(* PLC project Unnamed, Unknown Unnamed 1 *)
(* stored: creationDateTime 2025-11-24T11:16:17, modificationDateTime 2025-11-24T18:26:55 *)

PROGRAM Lab2
  VAR
    Potentiometer AT %IW1 : UINT := 0;
    Ljussensor AT %IW2 : UINT;
  END_VAR
  VAR
    S0 : BOOL := False;
    S1 : BOOL := False;
    Light_sample : BOOL := False;
    Poten_sample : BOOL;
    Light_damaged : BOOL := False;
    Poten_damaged : BOOL := False;
    Light_comp : UINT := 32768;
    Damaged : UINT := 0;
    High : UINT := 43690;
    Low : UINT := 21845;
  END_VAR
  VAR
    Relay AT %QX0.0 : BOOL := 0;
  END_VAR
  VAR
    CTU0 : CTU;
    TON0 : TON;
    T50ms : TIME := T#50ms;
    Tick_100ms : BOOL := 0;
    Fifty_ticks : INT := 50;
    TON1 : TON;
    R_TRIG0 : R_TRIG;
    F_TRIG0 : F_TRIG;
  END_VAR
  VAR  (* added by the conversion: wires and edge detectors of the diagram *)
    R_TRIG1 : R_TRIG;
    _GT34_OUT : BOOL;
    _LT35_OUT : BOOL;
    _EQ42_OUT : BOOL;
  END_VAR

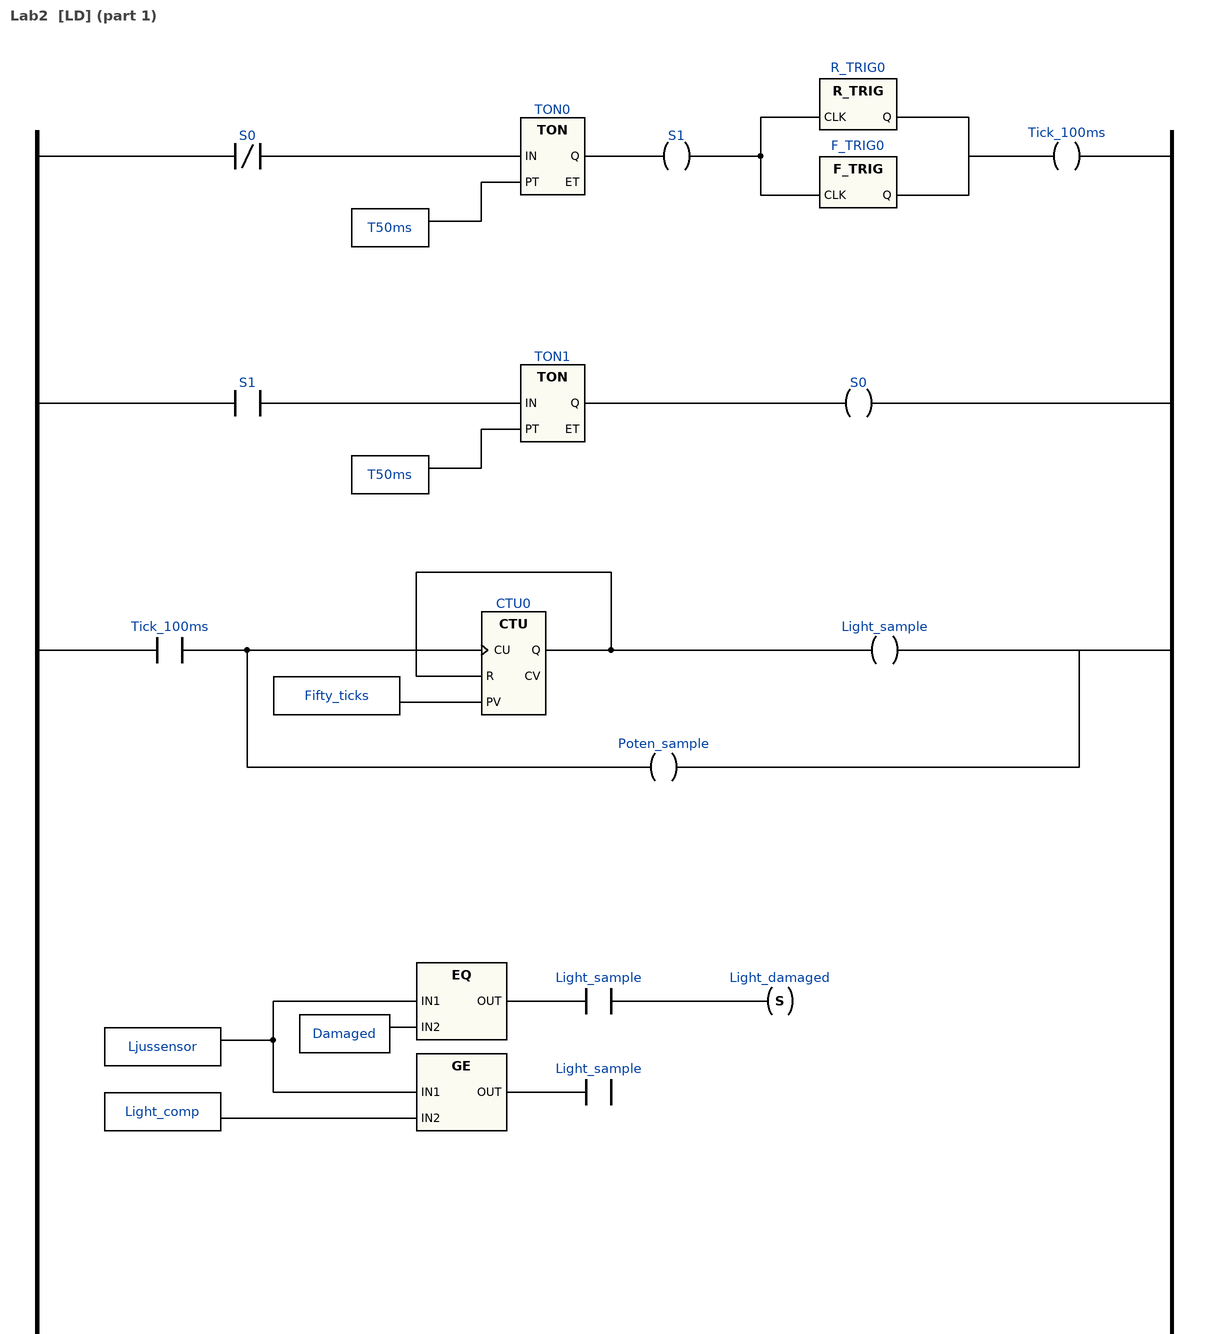
(* LD diagram, written out as Structured Text *)
TON0(IN := NOT S0, PT := T50ms);
R_TRIG0(CLK := TON0.Q);
F_TRIG0(CLK := TON0.Q);
Tick_100ms := R_TRIG0.Q OR F_TRIG0.Q;
R_TRIG1(CLK := Tick_100ms);
CTU0(CU := R_TRIG1.Q, R := CTU0.Q, PV := Fifty_ticks);
Light_sample := CTU0.Q;
TON1(IN := S1, PT := T50ms);
S0 := TON1.Q;
S1 := TON0.Q;
Poten_sample := Tick_100ms;
IF Ljussensor = Damaged AND Light_sample THEN Light_damaged := TRUE; END_IF;
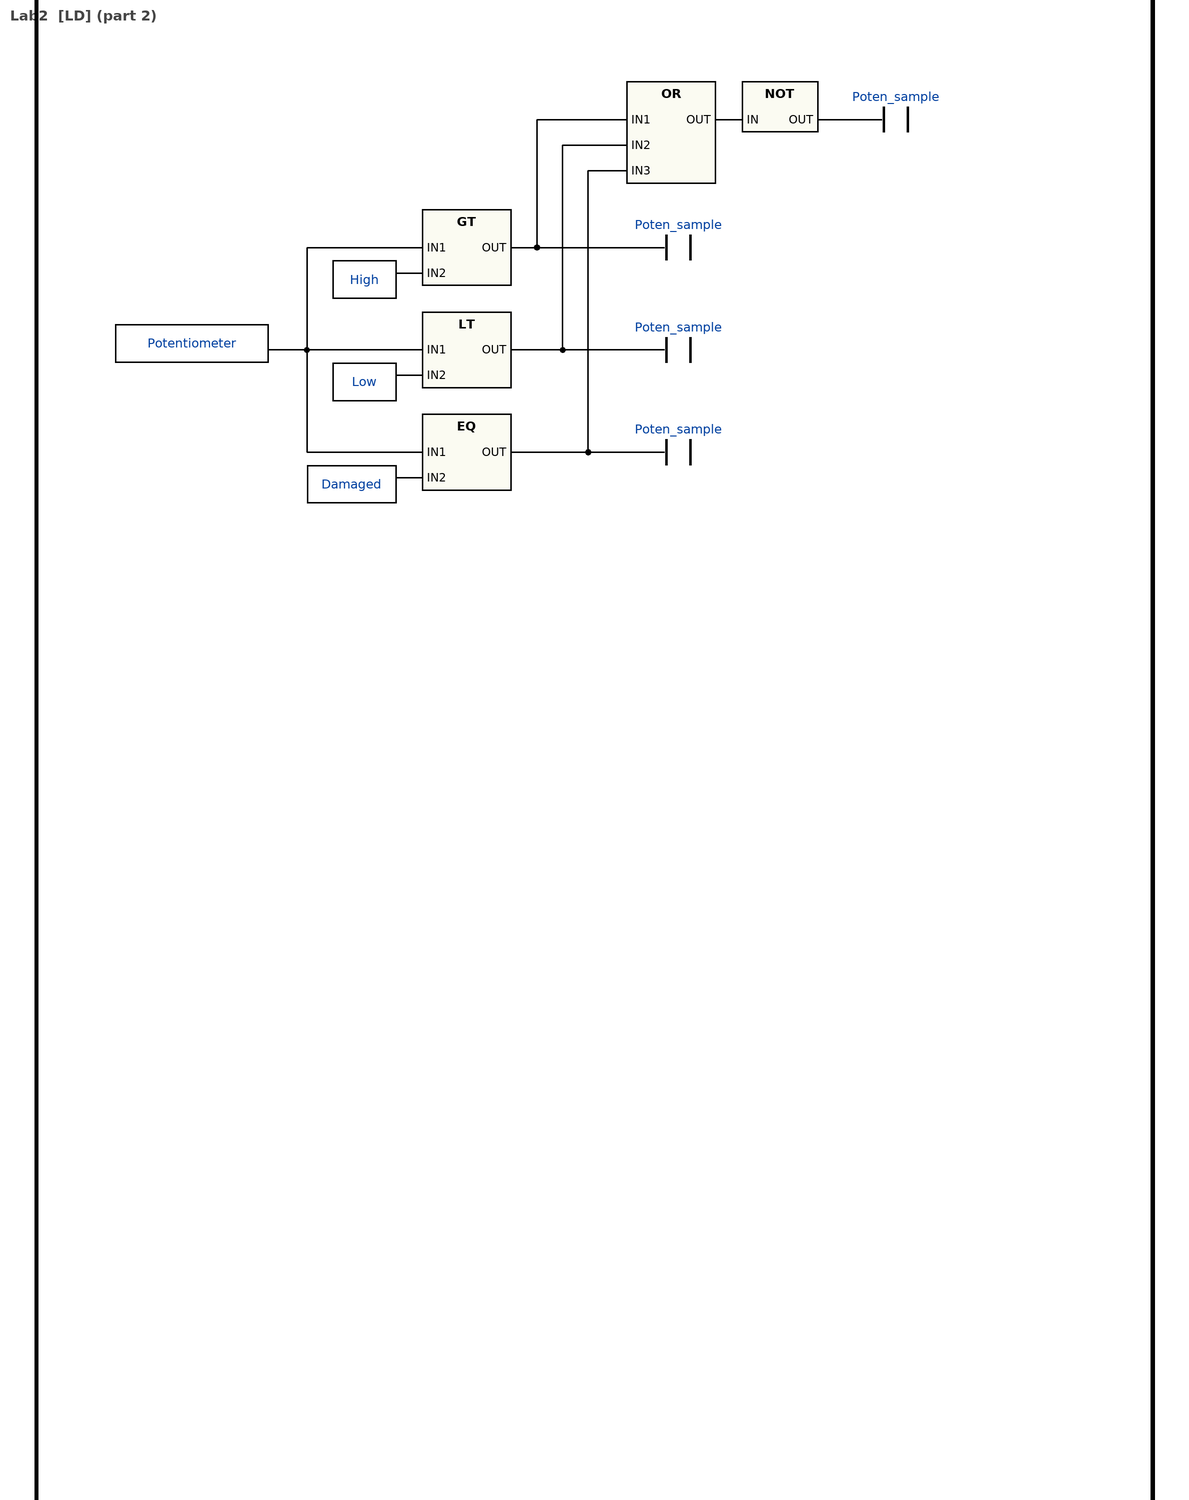
_GT34_OUT := Potentiometer > High;
_LT35_OUT := Potentiometer < Low;
_EQ42_OUT := Potentiometer = Damaged;
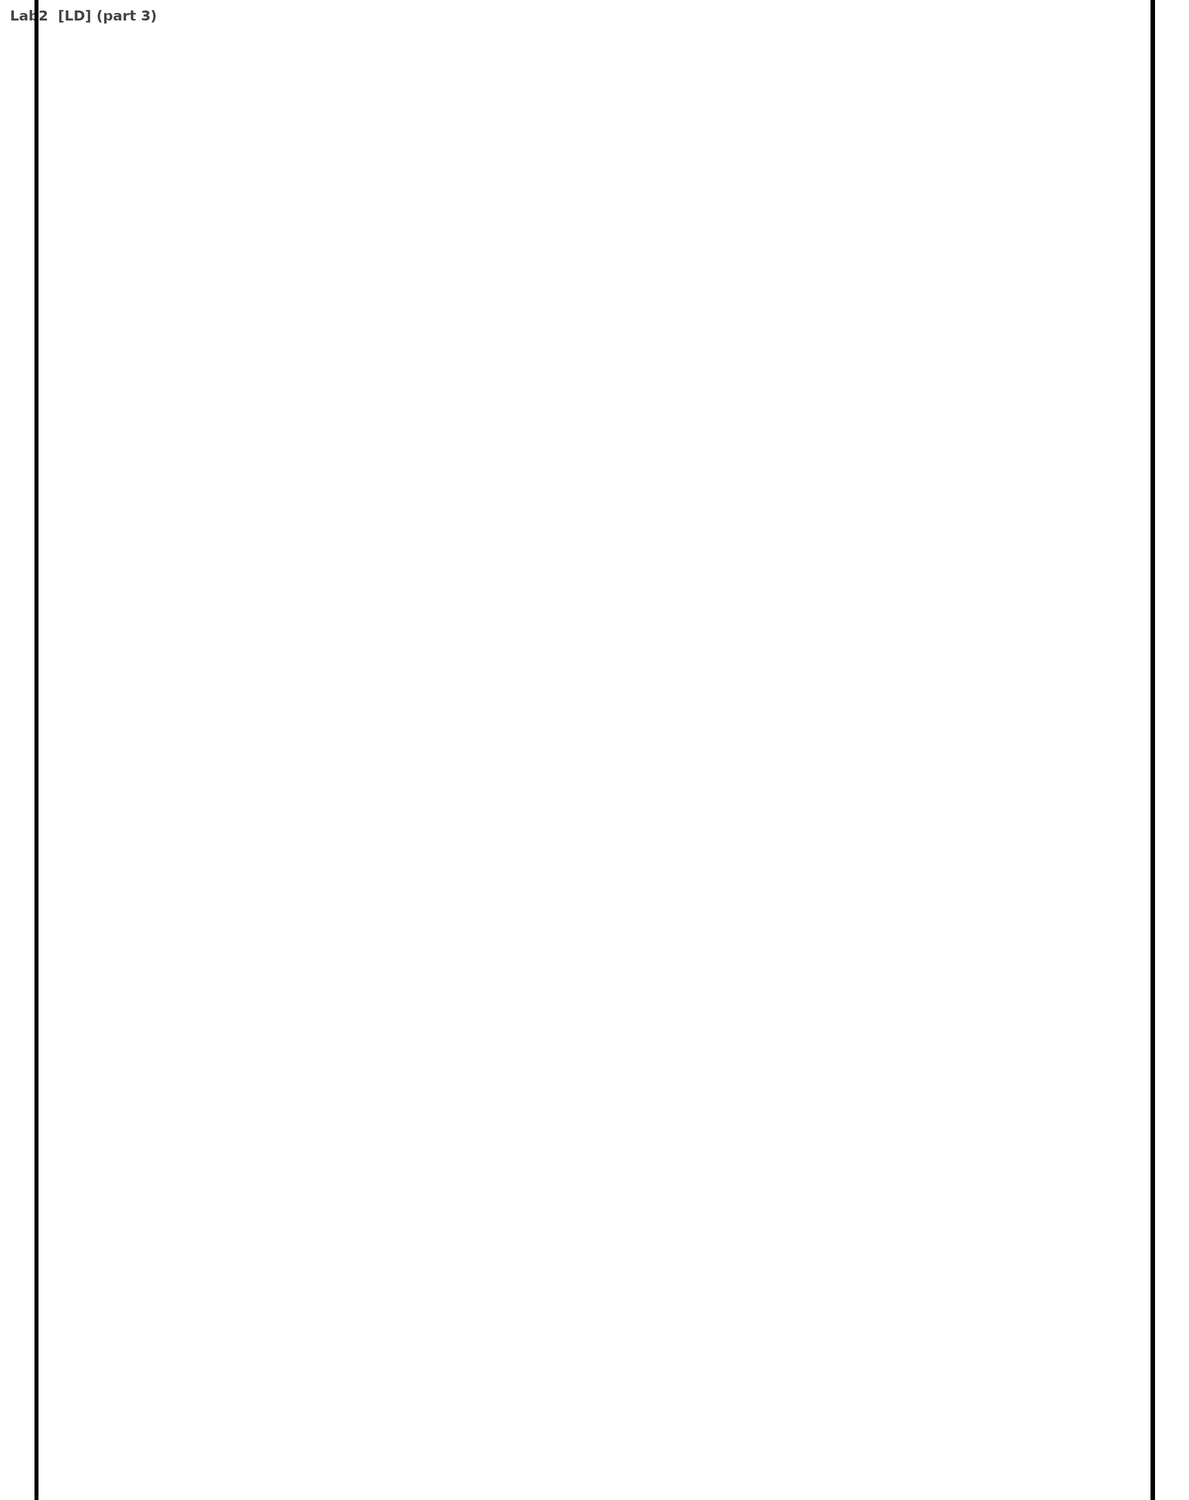
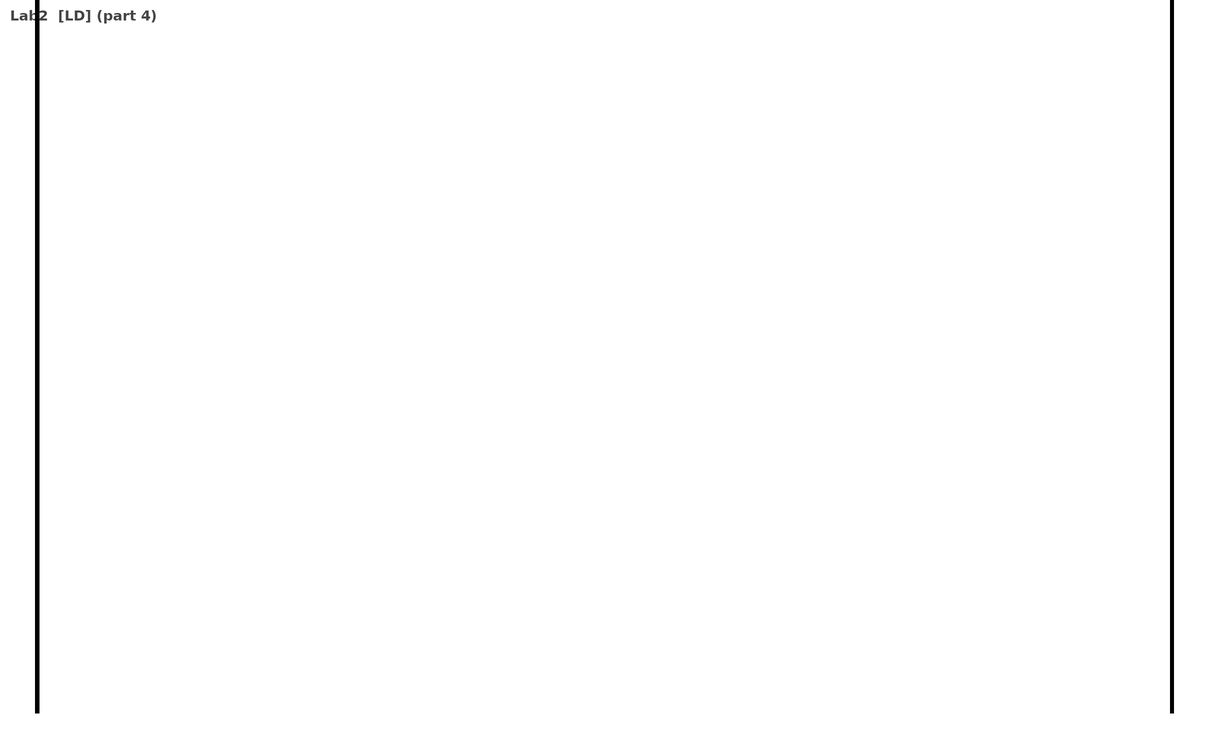
(* drawn but not wired to any output: Light_sample, Poten_sample, Poten_sample, Poten_sample, Poten_sample *)
END_PROGRAM

CONFIGURATION Config0
  RESOURCE Res0 ON PLC
    TASK task0(INTERVAL := T#20ms, PRIORITY := 0);
    PROGRAM instance0 WITH task0 : Lab2;
  END_RESOURCE
END_CONFIGURATION
